FUNCTION_BLOCK CentralServerControl (* Central Server Controller *)
  (* Standard: 61499-2 *)
  (* Version 0.2, 2003-12-04, JHC, Rockwell Automation, Renamed for better indexing. *)
  (* Version 0.1, 2002-11-05, JHC, Rockwell Automation, Corrected missing ST element in Algorithm REQ. *)
  (* Version 0.0, 2000-05-30, JHC, Rockwell Automation *)
  (* Compiler header: package fb.rt.cs725; *)
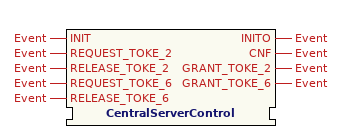
  EVENT_INPUT
    INIT; (* Initialization Request *)
    REQUEST_TOKE_2;
    RELEASE_TOKE_2;
    REQUEST_TOKE_6;
    RELEASE_TOKE_6;
  END_EVENT
  EVENT_OUTPUT
    INITO; (* Initialization Confirm *)
    CNF; (* Execution Confirmation *)
    GRANT_TOKE_2;
    GRANT_TOKE_6;
  END_EVENT
  VAR
    requestQueue : ARRAY [0..19] OF INT;
    arrayStart : INT;
    arrayEnd : INT;
    tokenAvailable : BOOL;
    tokenOwner : INT;
    targ2 : BOOL;
    targ6 : BOOL;
  END_VAR
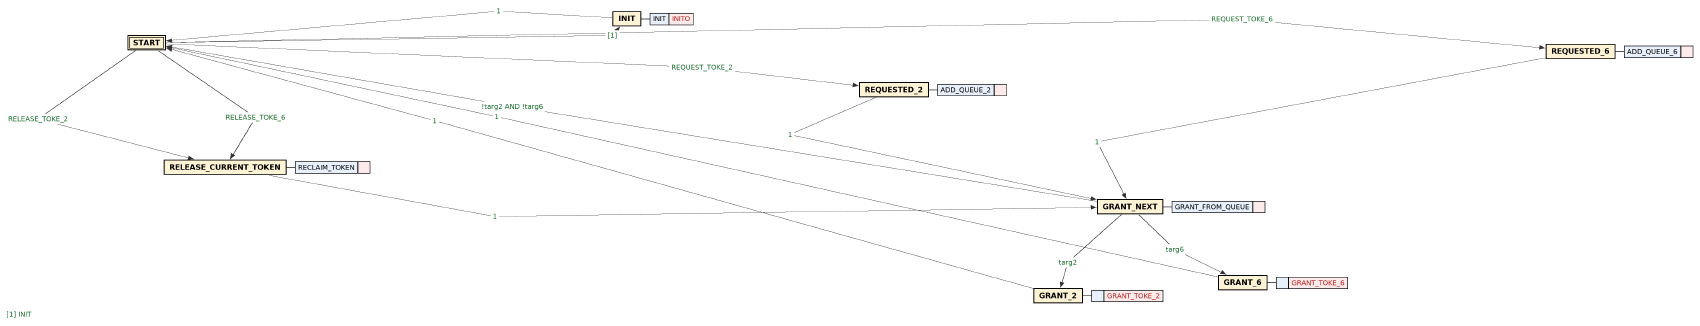
  EC_STATES
    START; (* Initial State *)
    INIT : INIT -> INITO; (* Initialization *)
    REQUESTED_2 : ADD_QUEUE_2;
    REQUESTED_6 : ADD_QUEUE_6;
    GRANT_NEXT : GRANT_FROM_QUEUE;
    RELEASE_CURRENT_TOKEN : RECLAIM_TOKEN;
    GRANT_2 : -> GRANT_TOKE_2;
    GRANT_6 : -> GRANT_TOKE_6;
  END_STATES
  EC_TRANSITIONS
    START TO INIT := INIT;
    INIT TO START := 1;
    START TO REQUESTED_6 := REQUEST_TOKE_6;
    START TO REQUESTED_2 := REQUEST_TOKE_2;
    REQUESTED_6 TO GRANT_NEXT := 1;
    REQUESTED_2 TO GRANT_NEXT := 1;
    GRANT_NEXT TO START := !targ2 AND !targ6;
    START TO RELEASE_CURRENT_TOKEN := RELEASE_TOKE_2;
    START TO RELEASE_CURRENT_TOKEN := RELEASE_TOKE_6;
    RELEASE_CURRENT_TOKEN TO GRANT_NEXT := 1;
    GRANT_NEXT TO GRANT_2 := targ2;
    GRANT_NEXT TO GRANT_6 := targ6;
    GRANT_6 TO START := 1;
    GRANT_2 TO START := 1;
  END_TRANSITIONS
  ALGORITHM INIT IN ST: (* Initialization algorithm *)
tokenAvailable := TRUE;
tokenOwner := 0;
arrayStart := 0;
arrayEnd := 0;
  END_ALGORITHM
  ALGORITHM REQ IN ST: (* Normally executed algorithm *)

  END_ALGORITHM
  ALGORITHM GRANT_FROM_QUEUE IN ST:
System.out.println("Entered queue granting algorithm");

//first check if the token is already taken
IF tokenAvailable = TRUE THEN

//if so, check if either position of the queue has a waiting requeust
    IF requestQueue[arrayStart] <> 0 THEN
        tokenAvailable := FALSE;
        tokenOwner := requestQueue[arrayStart];
        arrayStart := (arrayStart + 1) MOD 20;
    END_IF;

    IF tokenOwner = 2 THEN
        System.out.println("2");
    targ2 := TRUE;
    targ6 := FALSE;
    ELSIF tokenOwner = 6 THEN
        System.out.println("6");
    targ6 := TRUE;
    targ2 := FALSE;
    ELSE
        System.out.println("0");
    targ2 := FALSE;
    targ6 := FALSE;
    END_IF;

END_IF;
  END_ALGORITHM
  ALGORITHM RECLAIM_TOKEN IN ST:
tokenAvailable := TRUE;
tokenOwner := 0;
System.out.println("Token released and reclaimed!");
  END_ALGORITHM
  ALGORITHM ADD_QUEUE_2 IN ST:
requestQueue[arrayEnd] := 2;
arrayEnd := (arrayEnd + 1) MOD 20;
  END_ALGORITHM
  ALGORITHM ADD_QUEUE_6 IN ST:
requestQueue[arrayEnd] := 6;
arrayEnd := (arrayEnd + 1) MOD 20;
  END_ALGORITHM
END_FUNCTION_BLOCK
